PROGRAM MAIN
VAR
	bStartbutton : BOOL := FALSE;
	bStopbutton : BOOL := FALSE;

	bConveyoron : BOOL := FALSE;
END_VAR

bConveyoron := (bStartbutton OR bConveyoron) AND NOT bStopbutton;
IF bStartbutton := TRUE THEN
	bStopbutton := FALSE;
	bStartbutton := FALSE;
END_IF
IF bStopbutton := TRUE THEN
	bStopbutton := FALSE;
	bStartbutton := FALSE;
END_IF

END_PROGRAM

(* stored: Version 1.1.0.1, ProductVersion 3.1.4024.16
   POU MAIN: Id {1c53b36d-8f4a-4fc9-8da5-cec3460eb291}, SpecialFunc None *)
